// TIA Portal V18 export
ORGANIZATION_BLOCK "Emergency"   // OB31, LAD, CyclicInterrupt
{ S7_Optimized_Access := 'TRUE' }
VERSION : 0.1
// stored: AutoNumber true, IsIECCheckEnabled false, SetENOAutomatically false
   VAR_INPUT
      Initial_Call : Bool;   // Initial call of this OB
      Event_Count : Int;   // Events discarded
   END_VAR
BEGIN

REGION Network 1 (SCL): Checking ther conditions

   //1 FOR NO EMERGENCY, 0 IN CASE OF EMERGENCY
   //Only for the simulation, CAPACITIVE and PENDANT EMERGENCY should be added
   "Var".emergency_state := "emergency_mushroom";


   //Grounding is connected when it is 1 and 0 when it is not connected
   "Var".Grounding := "Ground_monitor_IBC" OR "Ground_monitor_truck";
END_REGION

REGION Network 2 (SCL): Defining kinds of unpredictable emergencies
   //Assign the emergencies

   // Emergency 1, fungo
   "Emergency_DB".Emergency_1 := NOT "emergency_mushroom";



   // Emergency 2, Pendant emergency
   "Emergency_DB".Emergency_2 := "Pendant_emergency_stop";



   // Emergency 3, Grounding
   "Emergency_DB".Emergency_3 := "Var".Grounding;



   // Emergency 4, HLS
   "Emergency_DB".Emergency_4 := "Capacitive_HLS";



   // Emergency 5, Temperature
   "Emergency_DB".Emergency_5 := NOT "Var".temperature_is_ok;



   // Emergency 6, NOT flow after 7 seconds OF In_loading state
   IF "Var".loading_flag THEN

       //signal of low flow, around 4mA, the value can be changed when we have connected the real FCV
       IF ABS("Flowmeter_analog" - 4) < 0.1 THEN

           //when it there is no flow, it starts a timer, if it remains the same for 7 seconds, shows an Emergency   
           "IEC_Timer_0_DB_5".TON(IN := "Var".loading_flag,
                                  PT := T#7S);



           IF "IEC_Timer_0_DB_5".Q THEN
               "Emergency_DB".Emergency_6 := 1;
           ELSE
               "Emergency_DB".Emergency_6 := 0;
           END_IF;

       END_IF;

   END_IF;
   // reseting the related timer
   IF NOT "Var".loading_flag THEN
       RESET_TIMER("IEC_Timer_0_DB_5"); 
   END_IF;



   "Var".no_flow_states := "Var".idle_flag OR "Var".emergency_flag OR "Var".pause_flag;
   // Emergency 7, Having flow in the idle Or pause state
   IF "Var".no_flow_states THEN

       "IEC_Timer_0_DB_11".TON(IN:="Var".no_flow_states,
                               PT:=T#3S);



       //If it is greater than the minimum (there is flow) after 3 seconds of being in Idle
       // the FLOW condition, can be changed! 
       IF "Flowmeter_analog" - 4 > 1 THEN


           IF "IEC_Timer_0_DB_11".Q THEN

               "Emergency_DB".Emergency_7 := 1;
           ELSE
               "Emergency_DB".Emergency_7 := 0;
           END_IF;


       END_IF;


   END_IF;
   //reseting the related timer
   IF NOT "Var".no_flow_states THEN
       RESET_TIMER("IEC_Timer_0_DB_11");
   END_IF;




   // Emergency 8, we are loading and FCV is closed
   IF "Var".loading_flag THEN

       //after 3 seconds being in loading and still the FCV is closed. 
       "IEC_Timer_0_DB_10".TON(IN:="Var".loading_flag,
                               PT:=T#3S);


       IF "IEC_Timer_0_DB_10".Q AND "FCV_valve_closed" THEN

           "Emergency_DB".Emergency_8 := 1;
       ELSE
           "Emergency_DB".Emergency_8 := 0;
       END_IF;

   END_IF;
   //reseting the timer in bellow



   // Emergency 9, we are in loading and ESD is closed
   IF "Var".loading_flag THEN

       //after 3 seconds being in loading and still the ESD is closed. 
       "IEC_Timer_0_DB_13".TON(IN := "Var".loading_flag,
                               PT := T#1500ms);




       IF "IEC_Timer_0_DB_13".Q AND "ESD_valve_closed" THEN

           "Emergency_DB".Emergency_9 := 1;
       ELSE
           "Emergency_DB".Emergency_9 := 0;
       END_IF;

   END_IF;
   //reseting the tiemrs
   IF NOT "Var".loading_flag THEN
       RESET_TIMER("IEC_Timer_0_DB_10");
       RESET_TIMER("IEC_Timer_0_DB_13");
   END_IF;
END_REGION
END_ORGANIZATION_BLOCK
